// TIA Portal V20 export
// export: Created 2026-07-16T12:58:46.2842904Z, ExportSetting WithDefaults, DisplayName Totally Integrated Automation Portal, DisplayVersion V20 Update 5, DisplayName TIA Portal Openness, DisplayVersion V20 Update 4, DisplayName TIA Portal Version Control Interface, DisplayVersion V20 Update 5, DisplayName SINAMICS Startdrive Advanced, DisplayVersion V20, DisplayName SINAMICS DCC, DisplayVersion V20, DisplayName SINAMICS Startdrive G130, G150, S120, S150, SINAMICS MV, G220, S200, S210, DisplayVersion V20, DisplayName SINAMICS Startdrive G110M, G120, G120C, G120D, G120P, G115D, DisplayVersion V20, DisplayName STEP 7 Professional, DisplayVersion V20 Update 5, DisplayName STEP 7 Safety, DisplayVersion V20 Update 2, DisplayName WinCC Basic/Comfort/Advanced, DisplayVersion V20 Update 5, DisplayName WinCC Unified, DisplayVersion V20 Update 5
DATA_BLOCK "DB_Settings"   // DB3
{ S7_Optimized_Access := 'TRUE' }
VERSION : 0.1
// Plant/system-level tunables (C-307) - HMI/operator writes, PLC read-only (C-308). Start values are commissioning defaults (C-309). Members with no start value shown are genuinely unconfigured pending real numbers from the project owner - see the presented build notes, not a guess.
// stored: AutoNumber true, DBAccessibleFromOPCUA true, IsOnlyStoredInLoadMemory false, IsRetainMemResEnabled false, IsWriteProtectedInAS false, MemoryReserve 100
   VAR RETAIN
      PreStartSounderTime : Real := 10.0;
      ShredderReverseRunTime : Real := 6.0;
      InfeedRestartDelay : Real := 5.0;
      InfeedToUpstreamEnableDelay : Real := 3.0;
      OvercurrentSetpointMedium : Real;
      OvercurrentSetpointHigh : Real;
      OvercurrentMediumDelay : Real;
      OvercurrentHighDelay : Real;
      OvercurrentSpinUpAllowance : Real := 3.0;
      ReversalRetryPauseTime : Real := 4.0;
      ReversalWindowTime : Real := 180.0;
      ReversalCountThreshold : Int := 5;
      PressureTripConfirmTime : Real := 0.5;
      PressureClearResumeDelay : Real;
      PressureTripCountThreshold : Int := 5;
      PusherEndTravelTimeout : Real;
      PusherParkedTimeout : Real;
      PusherEndTravelHoldTime : Real := 2.0;
      PusherPumpRunOnTime : Real;
      PusherJogWarningTime : Real := 1.0;
      PusherFitted : Bool := TRUE;
      DischargeConveyorTimeout : Real;
   END_VAR
BEGIN
END_DATA_BLOCK
